(* Logix 5000 project; controller ARS14002_PLC vendor 1 type 14 code 218 rev 30.11; software revision 30.01; part 6 of 13 *)
(* tags used below, declared in another part *)
   ARS_COLLECT : BOOL;
   ARS_COLLECT_AUTO : BOOL;
   ARS_DERIME_AUTO : BOOL;
   AT2_PLANT_ATOMIZING : BOOL;
   AT2_PLANT_BACKFILL : BOOL;
   AT2_PLANT_COLLECT_AUTO : BOOL;
   AT3_PLANT_ATOMIZING : BOOL;
   AT3_PLANT_BACKFILL : BOOL;
   AT3_PLANT_COLLECT_AUTO : BOOL;
   BACKFILL_PAUSE_BLOWBACK_ONS : BOOL;
   BLOWBACK_COMMAND : BOOL;
   BLOWBACK_COUNTER : COUNTER;
   BLOWBACK_PRESS_SPH : REAL;
   BLOWBACK_PRESS_SPL : REAL;
   BLOWBACK_PRESS_UNSAFE : REAL;
   BLOWBACK_REQUEST : BOOL;
   BLOWBACK_REQUEST_OFF_ONS : BOOL;
   BLOWBACK_REQUEST_ONS : BOOL;
   BLOWBACKS_REQUESTED : DINT;
   CALC_NEXT_MONTH_OSR_OB : BOOL;
   COLDBOX_IDLE : BOOL;
   COLDBOX_STANDBY : BOOL;
   Collect_Stop_Dew_Pt : BOOL;
   Collect_Stop_O2 : BOOL;
   FCV_101A : CM_AO_VLV;
   FCV_101B : CM_AO_VLV;
   FCV_101C : CM_AO_VLV;
   FCV_202 : CM_AO_VLV;
   FCV_202_BLOWBACK_POS : REAL;
   FCV_202_OPEN_DLA_PILOT_ADJ : DINT;
   FCV_202_OPEN_DLA_SEC : REAL;
   FCV_202_OPEN_DLA_TMR : TIMER;
   FCV_202_OPEN_INIT : TIMER;
   FCV_202_PVSWITCH : BOOL;   // 0 = PIT-201 1 = PIT-101C
   FCV_202_STARTPOS : REAL;
   FCV_204_ATOMIZE_INIT : TIMER;
   FCV_207_BLOWOFF : BOOL;
   FCV_207_FRONT_END_RESCUE : BOOL;
   FCV_207_FRONT_END_RESCUE_AUTO : BOOL;
   FCV_207_FRONT_END_RESCUE_SP : REAL;
   FCV_207_POSTHEAT_OFF : BOOL;   // Turn off 207 post heat pressurizing
   FCV_207_POSTHEATPRESSURE : REAL;
   FCV_207_POSTHEATPRESSURE_DB : REAL;
   FCV_207_PRESSRELIEF_SPH : REAL;
   FCV_207_PRESSRELIEF_SPL : REAL;
   FCV_207_STATICPOS : REAL;
   FCV_504_LOWPRESS_MAXOPEN : REAL;
   FCV_504_PT_603_LOLOALM : BOOL;
   FCV_504_PT_603_LOWALM : BOOL;
   FCV_504_PT_603_LOWLIM : REAL;
   FCV_504_PT_603_LOWLIM_RESET : REAL;
   FCV_504_SP_Atomize : REAL;
   FCV_504_SP_Atomize_2Tower : REAL;
   FCV_504_SP_Atomize_2Tower_AR : REAL;
   FCV_504_SP_Atomize_2Tower_AR_CALC : REAL;
   FCV_504_SP_Atomize_2Tower_CALC : REAL;
   FCV_504_SP_Atomize_AR : REAL;
   FCV_504_SP_Atomize_AR_CALC : REAL;   // Setpoint with an adjustment for the Pilot Plant
   FCV_504_SP_Atomize_AR_PILOT_ADJ : REAL;   // Adjustment for the atomize setpoint on top of what it would be for normal furnaces
   FCV_504_SP_Atomize_CALC : REAL;
   FCV_504_SP_Atomize_FRONT_END : REAL;
   FCV_504_SP_Atomize_PILOT_ADJ : REAL;
   FCV_504_SP_Idle : REAL;
   FCV_504_SP_Idle_AR : REAL;
   FCV_504_SP_Idle_AR_STORAGE : REAL;
   FCV_504_SP_Idle_STORAGE : REAL;
   FCV_504_SP_Standby : REAL;
   FCV_504_SP_Standby_AR : REAL;
   FCV_504_STARTPOS : REAL;
   FCV_603_Atomize_Start_CV : REAL;
   FCV_603_BUMP_TMR : TIMER;
   FCV_603_SP_Atomize : REAL;
   FCV_603_SP_Idle : REAL;
   FCV_603_SP_Standby : REAL;
   MODE_ATOMIZE : BOOL;
   MODE_IDLE : BOOL;
   MODE_STANDBY_IDLE : BOOL;
   MODE_STANDBY_PUMPUP : BOOL;
   PDT_603 : CM_AI_SCL_ALT;
   PDT_701 : CM_AI_SCL_ALT;
   PIDE_202 : PID_ENHANCED;
   PIDE_204 : PID_ENHANCED;
   PIDE_207 : PID_ENHANCED;
   PIDE_504 : PID_ENHANCED;
   PIDE_504_FRONT_END_CONTROL : BOOL;
   PIDE_504_FRONT_END_CONTROL_REQUEST : BOOL;
   PIDE_504_MODE : BOOL;   // 0 = Argon (PT-601) 1 = N2 (PT-603)
   PIDE_603 : PID_ENHANCED;
   PIDE_603_CVLimit_TON : TIMER;
   PIDE_603_CVLimitLOW_TON : TIMER;
   PIDE_605 : PID_ENHANCED;
   Pilot_Atomizing_Valve_Close_TON : TIMER;
   Pilot_Atomizing_Valve_Open_TON : TIMER;
   Pilot_Inlet_Valve_Open_TON : TIMER;
   PILOT_PLANT_ATOMIZING : BOOL;
   PILOT_PLANT_BACKFILL : BOOL;
   PILOT_PLANT_COLLECT_AUTO : BOOL;
   PT_1002 : CM_AI_SCL;
   PT_101C : CM_AI_SCL;
   PT_201 : CM_AI_SCL;
   PT_222 : CM_AI_SCL;
   PT_601 : CM_AI_SCL;
   PT_601_FCV_202_SP : REAL;
   PT_601_LR : CM_AI_SCL;
   PT_603 : CM_AI_SCL;
   Pull_Hold : BOOL;
   PWHMI_Post_Atomize_TMR : TIMER;
   SV_202F : CM_DO_GENERIC;
   SV_205 : CM_DO_GENERIC;
   SV_205_FIXED : BOOL;
   SV_205_Pressure_SPH : REAL;
   SV_205_Pressure_SPH_TEST : REAL;
   SV_205_Pressure_SPL : REAL;
   SV_205_Pressure_SPL_TEST : REAL;
   SV_207F : CM_DO_GENERIC;
   SV_221X : CM_DO_GENERIC;
   SV_221X_ONS : BOOL;
   SV_504F : CM_DO_GENERIC;
   SV_505X : CM_DO_GENERIC;
   SV_603F : CM_DO_GENERIC;
   SV_605F : CM_DO_GENERIC;
   TE_501 : CM_AI_SCL;
   TE_501_MIN_SV_202 : REAL;
   TE_902 : CM_AI_SCL;
   TimeStamp : DINT[7];
   TK_220_FILLS_MONTH : COUNTER;
   TK_220_Pressure_SPH : INT;
   TK_220_Pressure_SPL : INT;
   TK_700_Full : BOOL;
   TK_700_FULL_DLA_TMR : TIMER;
   TK_700_Full_SPH : REAL;
   TK_700_Full_SPL : REAL;
   TK_700_Low : BOOL;
   TK_700_LOW_DLA_TMR : TIMER;
   TK_700_Low_SPH : REAL;
   TK_700_Low_SPL : REAL;
   TK_700_NOT_FULL_DLA_TMR : TIMER;
   TK_700_OVERFULL_DLA_TMR : TIMER;
   XV_505_PT_603_SPH_VENT : REAL;
   XV_505_PT_603_SPL_VENT : REAL;
(* MainProgram, continued *)

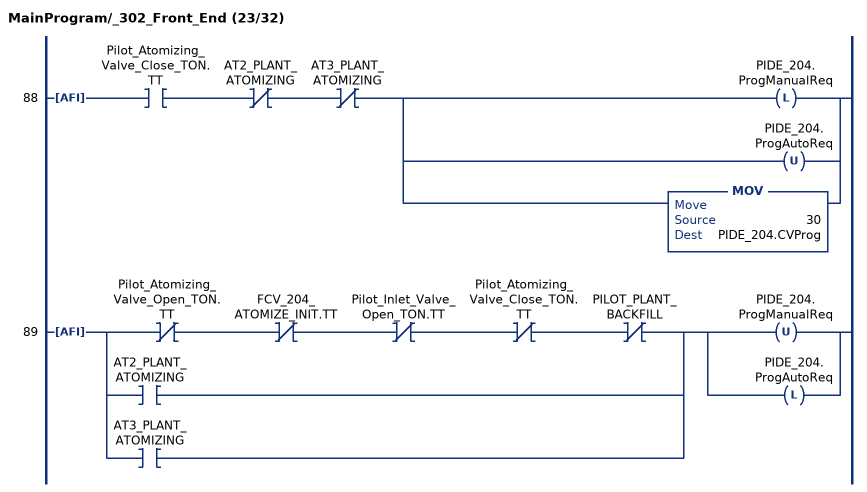
   [picture p107: MainProgram/_302_Front_End rungs 88-89]
   88: AFI()XIC(Pilot_Atomizing_Valve_Close_TON.TT)XIO(AT2_PLANT_ATOMIZING)XIO(AT3_PLANT_ATOMIZING)[OTL(PIDE_204.ProgManualReq) ,OTU(PIDE_204.ProgAutoReq) ,MOV(30,PIDE_204.CVProg) ];
   89: AFI()[XIO(Pilot_Atomizing_Valve_Open_TON.TT) XIO(FCV_204_ATOMIZE_INIT.TT) XIO(Pilot_Inlet_Valve_Open_TON.TT) XIO(Pilot_Atomizing_Valve_Close_TON.TT) XIO(PILOT_PLANT_BACKFILL) ,XIC(AT2_PLANT_ATOMIZING) ,XIC(AT3_PLANT_ATOMIZING) ][OTU(PIDE_204.ProgManualReq) ,OTL(PIDE_204.ProgAutoReq) ];
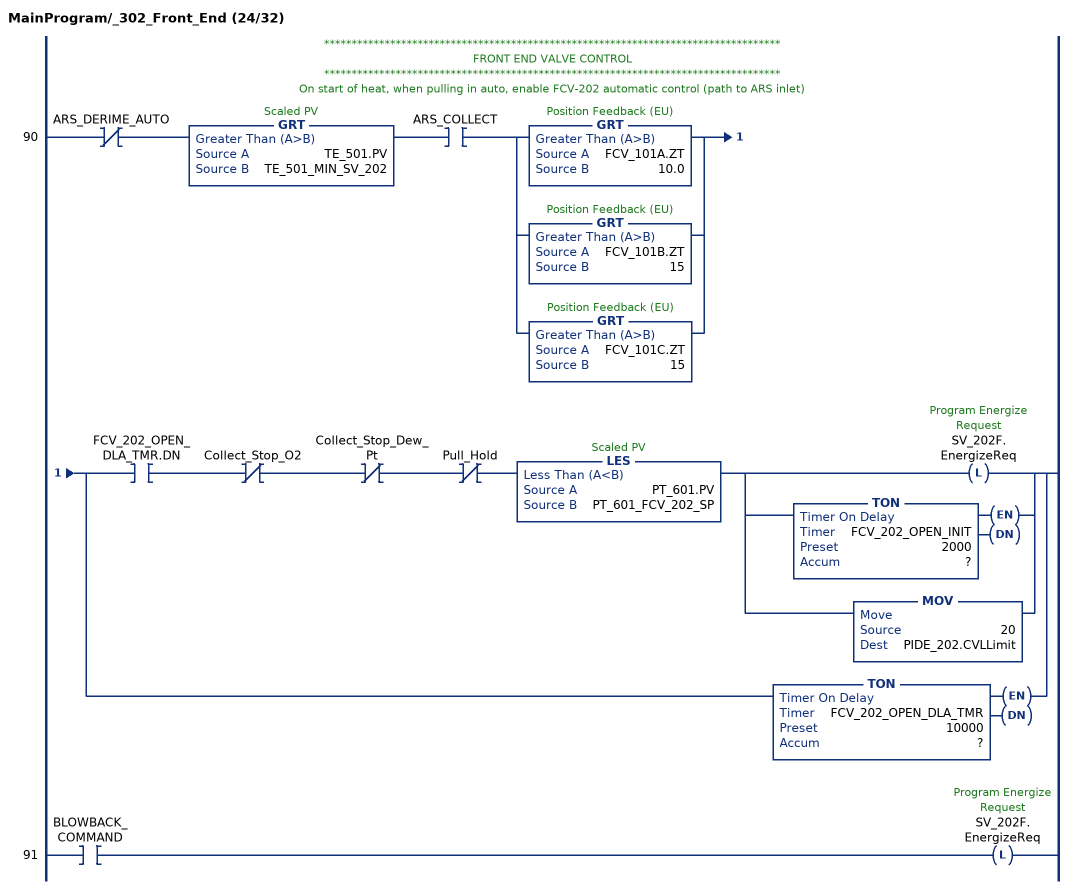
   // ***********************************************************************************
   // FRONT END VALVE CONTROL
   // ***********************************************************************************
   // On start of heat, when pulling in auto, enable FCV-202 automatic control (path to ARS inlet)
   90: XIO(ARS_DERIME_AUTO)GRT(TE_501.PV,TE_501_MIN_SV_202)XIC(ARS_COLLECT)[GRT(FCV_101A.ZT,10.0) ,GRT(FCV_101B.ZT,15) ,GRT(FCV_101C.ZT,15) ][XIC(FCV_202_OPEN_DLA_TMR.DN) XIO(Collect_Stop_O2) XIO(Collect_Stop_Dew_Pt) XIO(Pull_Hold) LES(PT_601.PV,PT_601_FCV_202_SP) [OTL(SV_202F.EnergizeReq) ,TON(FCV_202_OPEN_INIT,?,?) ,MOV(20,PIDE_202.CVLLimit) ] ,TON(FCV_202_OPEN_DLA_TMR,?,?) ];
   91: XIC(BLOWBACK_COMMAND)OTL(SV_202F.EnergizeReq);
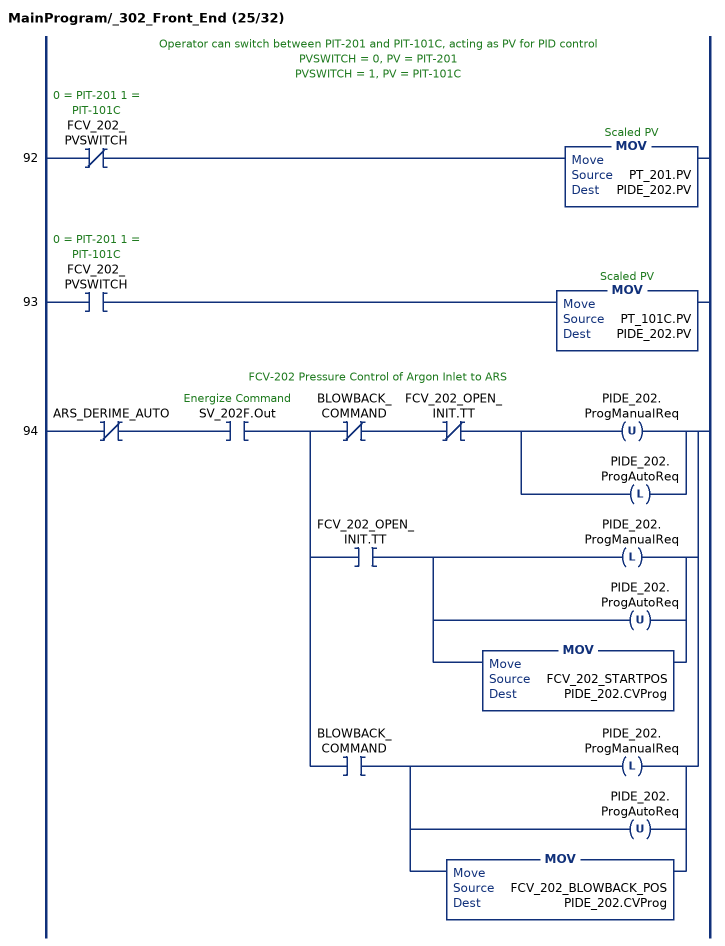
   // Operator can switch between PIT-201 and PIT-101C, acting as PV for PID control
   // PVSWITCH = 0, PV = PIT-201
   // PVSWITCH = 1, PV = PIT-101C
   92: XIO(FCV_202_PVSWITCH)MOV(PT_201.PV,PIDE_202.PV);
   93: XIC(FCV_202_PVSWITCH)MOV(PT_101C.PV,PIDE_202.PV);
   // FCV-202 Pressure Control of Argon Inlet to ARS
   94: XIO(ARS_DERIME_AUTO)XIC(SV_202F.Out)[XIO(BLOWBACK_COMMAND) XIO(FCV_202_OPEN_INIT.TT) [OTU(PIDE_202.ProgManualReq) ,OTL(PIDE_202.ProgAutoReq) ] ,XIC(FCV_202_OPEN_INIT.TT) [OTL(PIDE_202.ProgManualReq) ,OTU(PIDE_202.ProgAutoReq) ,MOV(FCV_202_STARTPOS,PIDE_202.CVProg) ] ,XIC(BLOWBACK_COMMAND) [OTL(PIDE_202.ProgManualReq) ,OTU(PIDE_202.ProgAutoReq) ,MOV(FCV_202_BLOWBACK_POS,PIDE_202.CVProg) ] ];
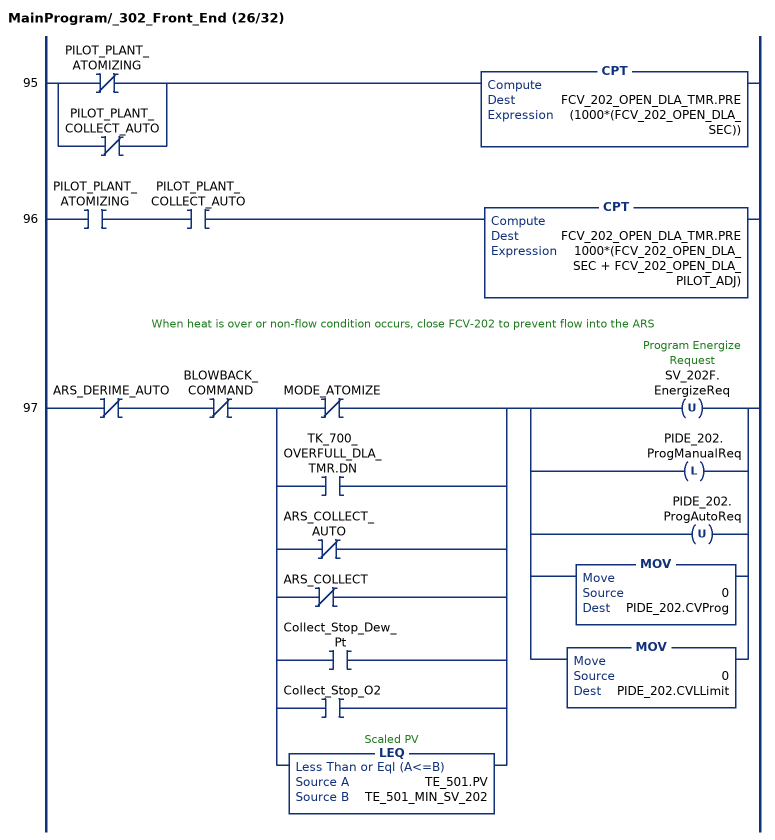
   95: [XIO(PILOT_PLANT_ATOMIZING) ,XIO(PILOT_PLANT_COLLECT_AUTO) ]CPT(FCV_202_OPEN_DLA_TMR.PRE,(1000*(FCV_202_OPEN_DLA_SEC)));
   96: XIC(PILOT_PLANT_ATOMIZING)XIC(PILOT_PLANT_COLLECT_AUTO)CPT(FCV_202_OPEN_DLA_TMR.PRE,1000*(FCV_202_OPEN_DLA_SEC + FCV_202_OPEN_DLA_PILOT_ADJ));
   // When heat is over or non-flow condition occurs, close FCV-202 to prevent flow into the ARS
   97: XIO(ARS_DERIME_AUTO)XIO(BLOWBACK_COMMAND)[XIO(MODE_ATOMIZE) ,XIC(TK_700_OVERFULL_DLA_TMR.DN) ,XIO(ARS_COLLECT_AUTO) ,XIO(ARS_COLLECT) ,XIC(Collect_Stop_Dew_Pt) ,XIC(Collect_Stop_O2) ,LEQ(TE_501.PV,TE_501_MIN_SV_202) ][OTU(SV_202F.EnergizeReq) ,OTL(PIDE_202.ProgManualReq) ,OTU(PIDE_202.ProgAutoReq) ,MOV(0,PIDE_202.CVProg) ,MOV(0,PIDE_202.CVLLimit) ];
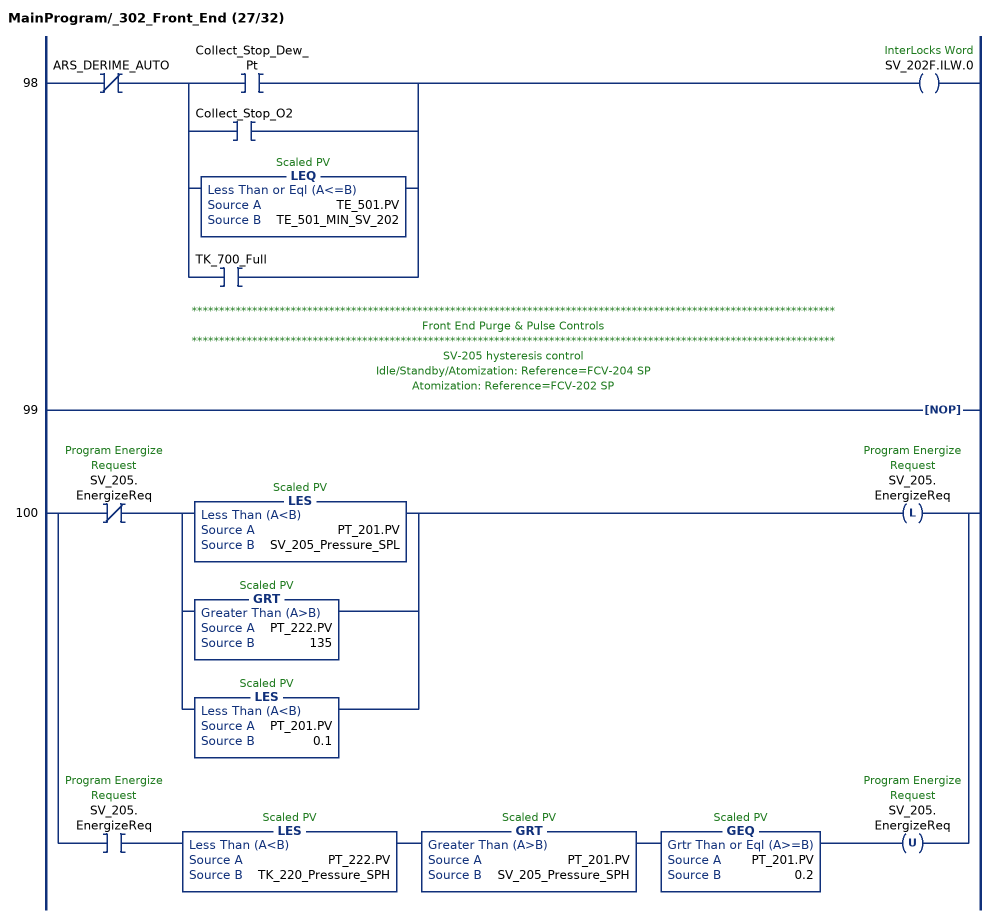
   98: XIO(ARS_DERIME_AUTO)[XIC(Collect_Stop_Dew_Pt) ,XIC(Collect_Stop_O2) ,LEQ(TE_501.PV,TE_501_MIN_SV_202) ,XIC(TK_700_Full) ]OTE(SV_202F.ILW.0);
   // *********************************************************************************************************************
   // Front End Purge & Pulse Controls
   // *********************************************************************************************************************
   // SV-205 hysteresis control
   // Idle/Standby/Atomization: Reference=FCV-204 SP
   // Atomization: Reference=FCV-202 SP
   99: NOP();
   100: [XIO(SV_205.EnergizeReq) [LES(PT_201.PV,SV_205_Pressure_SPL) ,GRT(PT_222.PV,135) ,LES(PT_201.PV,0.1) ] OTL(SV_205.EnergizeReq) ,XIC(SV_205.EnergizeReq) LES(PT_222.PV,TK_220_Pressure_SPH) GRT(PT_201.PV,SV_205_Pressure_SPH) GEQ(PT_201.PV,0.2) OTU(SV_205.EnergizeReq) ];
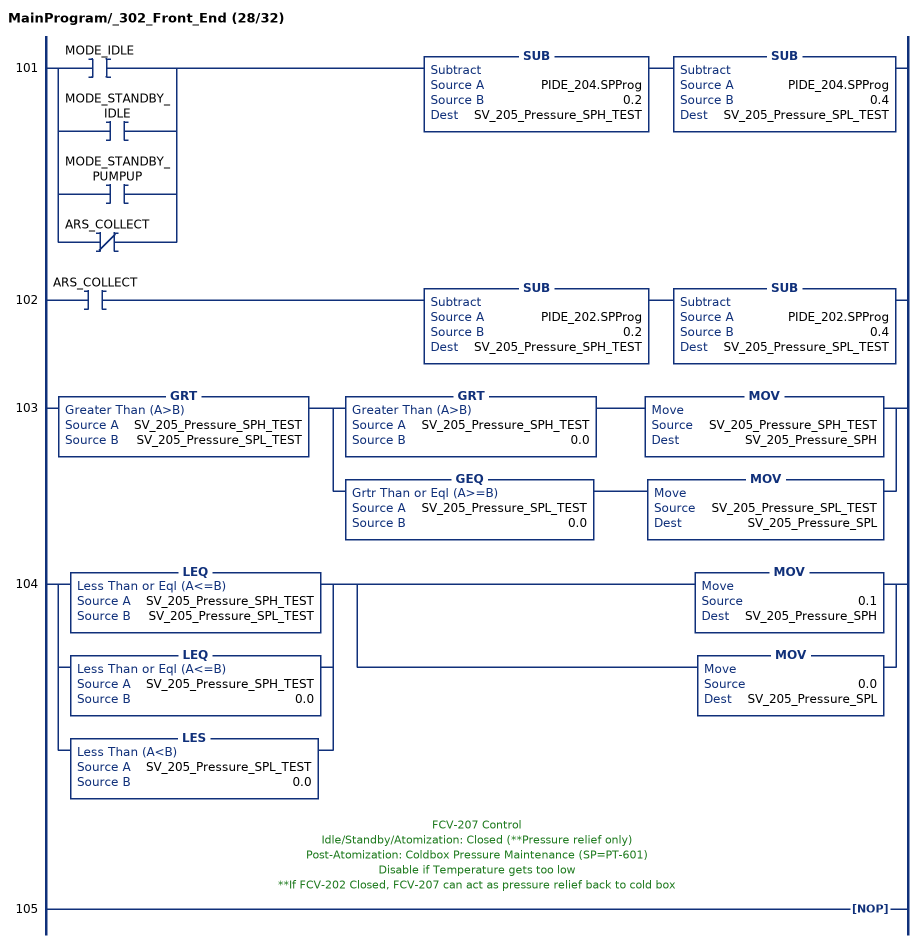
   101: [XIC(MODE_IDLE) ,XIC(MODE_STANDBY_IDLE) ,XIC(MODE_STANDBY_PUMPUP) ,XIO(ARS_COLLECT) ]SUB(PIDE_204.SPProg,0.2,SV_205_Pressure_SPH_TEST)SUB(PIDE_204.SPProg,0.4,SV_205_Pressure_SPL_TEST);
   102: XIC(ARS_COLLECT)SUB(PIDE_202.SPProg,0.2,SV_205_Pressure_SPH_TEST)SUB(PIDE_202.SPProg,0.4,SV_205_Pressure_SPL_TEST);
   103: GRT(SV_205_Pressure_SPH_TEST,SV_205_Pressure_SPL_TEST)[GRT(SV_205_Pressure_SPH_TEST,0.0) MOV(SV_205_Pressure_SPH_TEST,SV_205_Pressure_SPH) ,GEQ(SV_205_Pressure_SPL_TEST,0.0) MOV(SV_205_Pressure_SPL_TEST,SV_205_Pressure_SPL) ];
   104: [LEQ(SV_205_Pressure_SPH_TEST,SV_205_Pressure_SPL_TEST) ,LEQ(SV_205_Pressure_SPH_TEST,0.0) ,LES(SV_205_Pressure_SPL_TEST,0.0) ][MOV(0.1,SV_205_Pressure_SPH) ,MOV(0.0,SV_205_Pressure_SPL) ];
   // FCV-207 Control
   // Idle/Standby/Atomization: Closed (**Pressure relief only)
   // Post-Atomization: Coldbox Pressure Maintenance (SP=PT-601)
   // Disable if Temperature gets too low
   // **If FCV-202 Closed, FCV-207 can act as pressure relief back to cold box
   105: NOP();
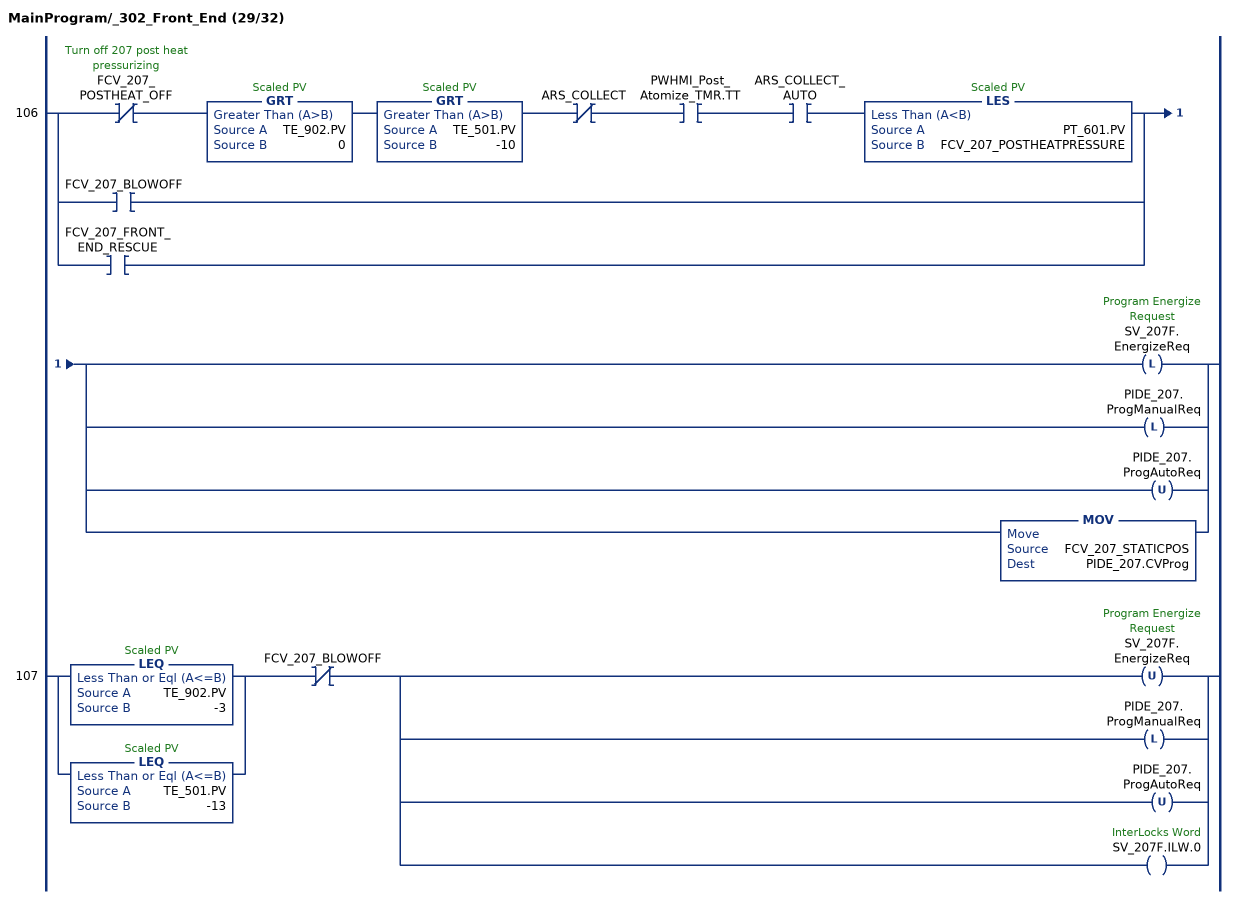
   106: [XIO(FCV_207_POSTHEAT_OFF) GRT(TE_902.PV,0) GRT(TE_501.PV,-10) XIO(ARS_COLLECT) XIC(PWHMI_Post_Atomize_TMR.TT) XIC(ARS_COLLECT_AUTO) LES(PT_601.PV,FCV_207_POSTHEATPRESSURE) ,XIC(FCV_207_BLOWOFF) ,XIC(FCV_207_FRONT_END_RESCUE) ][OTL(SV_207F.EnergizeReq) ,OTL(PIDE_207.ProgManualReq) ,OTU(PIDE_207.ProgAutoReq) ,MOV(FCV_207_STATICPOS,PIDE_207.CVProg) ];
   107: [LEQ(TE_902.PV,-3) ,LEQ(TE_501.PV,-13) ]XIO(FCV_207_BLOWOFF)[OTU(SV_207F.EnergizeReq) ,OTL(PIDE_207.ProgManualReq) ,OTU(PIDE_207.ProgAutoReq) ,OTE(SV_207F.ILW.0) ];
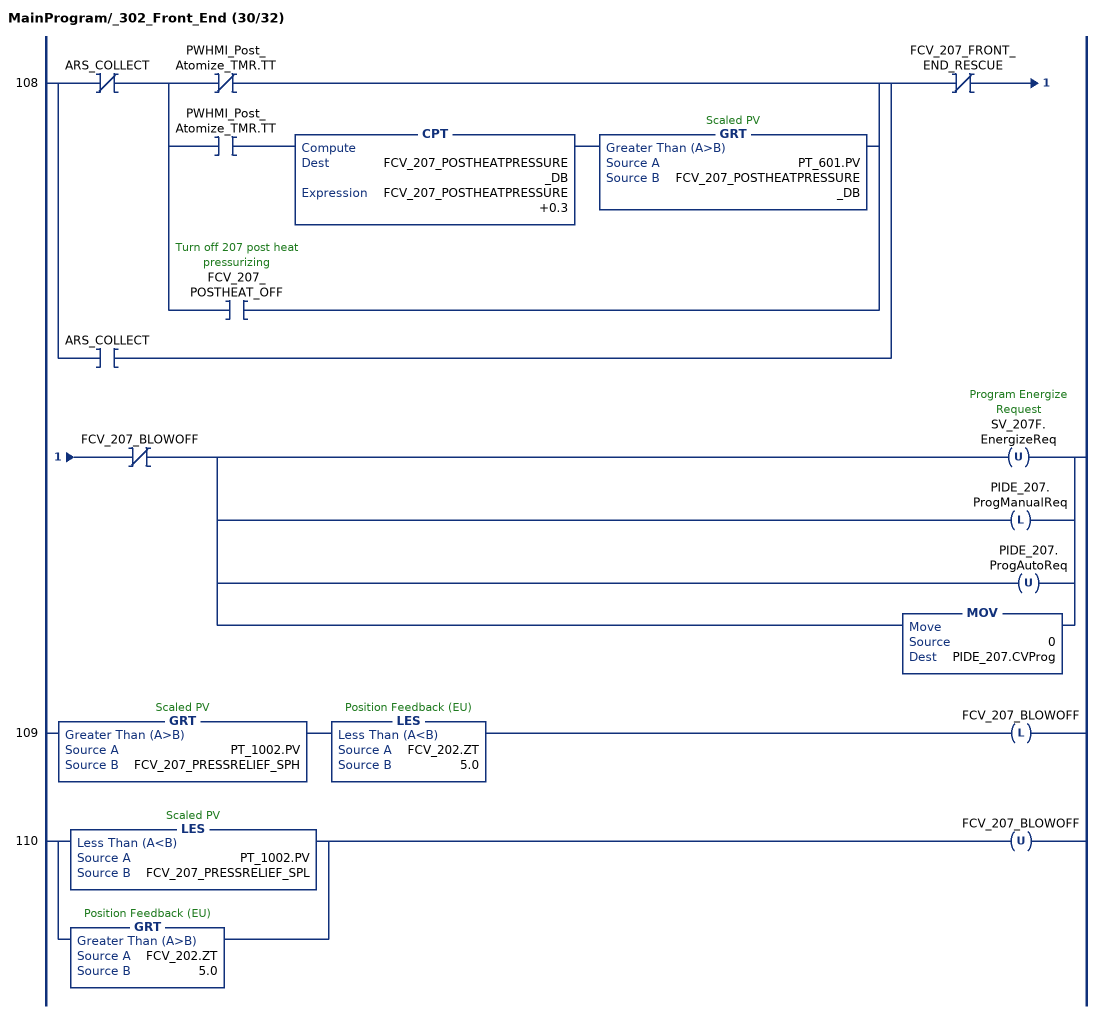
   108: [XIO(ARS_COLLECT) [XIO(PWHMI_Post_Atomize_TMR.TT) ,XIC(PWHMI_Post_Atomize_TMR.TT) CPT(FCV_207_POSTHEATPRESSURE_DB,FCV_207_POSTHEATPRESSURE+0.3) GRT(PT_601.PV,FCV_207_POSTHEATPRESSURE_DB) ,XIC(FCV_207_POSTHEAT_OFF) ] ,XIC(ARS_COLLECT) ]XIO(FCV_207_FRONT_END_RESCUE)XIO(FCV_207_BLOWOFF)[OTU(SV_207F.EnergizeReq) ,OTL(PIDE_207.ProgManualReq) ,OTU(PIDE_207.ProgAutoReq) ,MOV(0,PIDE_207.CVProg) ];
   109: GRT(PT_1002.PV,FCV_207_PRESSRELIEF_SPH)LES(FCV_202.ZT,5.0)OTL(FCV_207_BLOWOFF);
   110: [LES(PT_1002.PV,FCV_207_PRESSRELIEF_SPL) ,GRT(FCV_202.ZT,5.0) ]OTU(FCV_207_BLOWOFF);
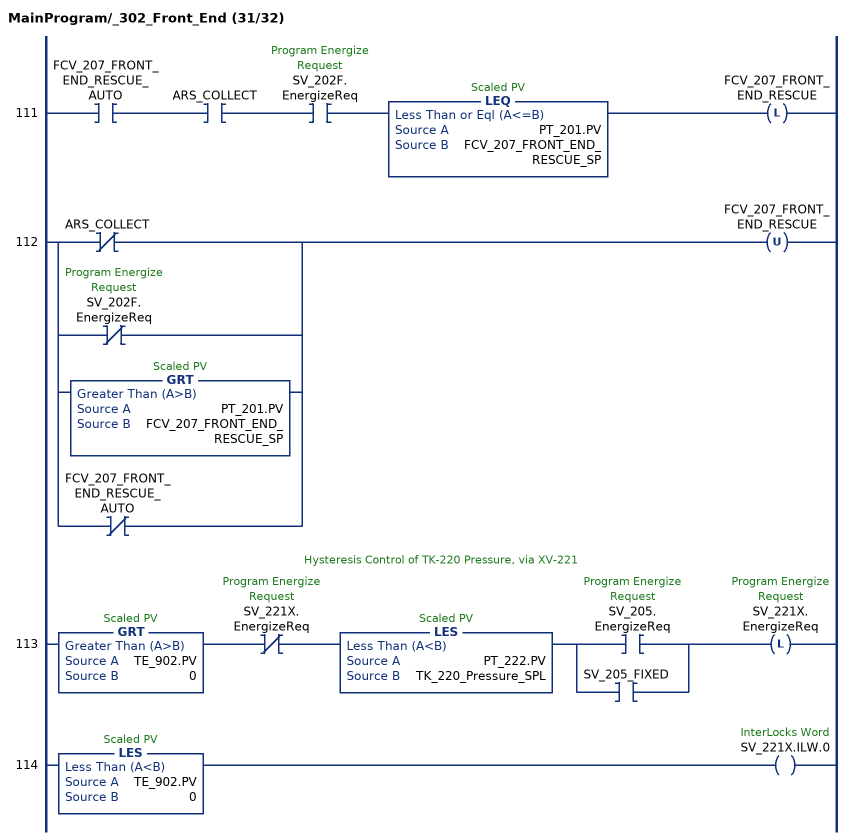
   111: XIC(FCV_207_FRONT_END_RESCUE_AUTO)XIC(ARS_COLLECT)XIC(SV_202F.EnergizeReq)LEQ(PT_201.PV,FCV_207_FRONT_END_RESCUE_SP)OTL(FCV_207_FRONT_END_RESCUE);
   112: [XIO(ARS_COLLECT) ,XIO(SV_202F.EnergizeReq) ,GRT(PT_201.PV,FCV_207_FRONT_END_RESCUE_SP) ,XIO(FCV_207_FRONT_END_RESCUE_AUTO) ]OTU(FCV_207_FRONT_END_RESCUE);
   // Hysteresis Control of TK-220 Pressure, via XV-221
   113: GRT(TE_902.PV,0)XIO(SV_221X.EnergizeReq)LES(PT_222.PV,TK_220_Pressure_SPL)[XIC(SV_205.EnergizeReq) ,XIC(SV_205_FIXED) ]OTL(SV_221X.EnergizeReq);
   114: LES(TE_902.PV,0)OTE(SV_221X.ILW.0);
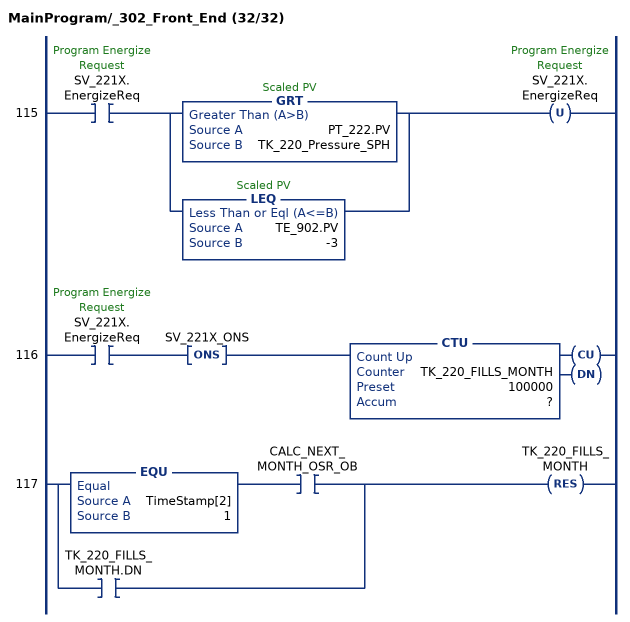
   115: XIC(SV_221X.EnergizeReq)[GRT(PT_222.PV,TK_220_Pressure_SPH) ,LEQ(TE_902.PV,-3) ]OTU(SV_221X.EnergizeReq);
   116: XIC(SV_221X.EnergizeReq)ONS(SV_221X_ONS)CTU(TK_220_FILLS_MONTH,?,?);
   117: [EQU(TimeStamp[2],1) XIC(CALC_NEXT_MONTH_OSR_OB) ,XIC(TK_220_FILLS_MONTH.DN) ]RES(TK_220_FILLS_MONTH);
END_ROUTINE

ROUTINE _303_Cold_Box   (* ladder *)
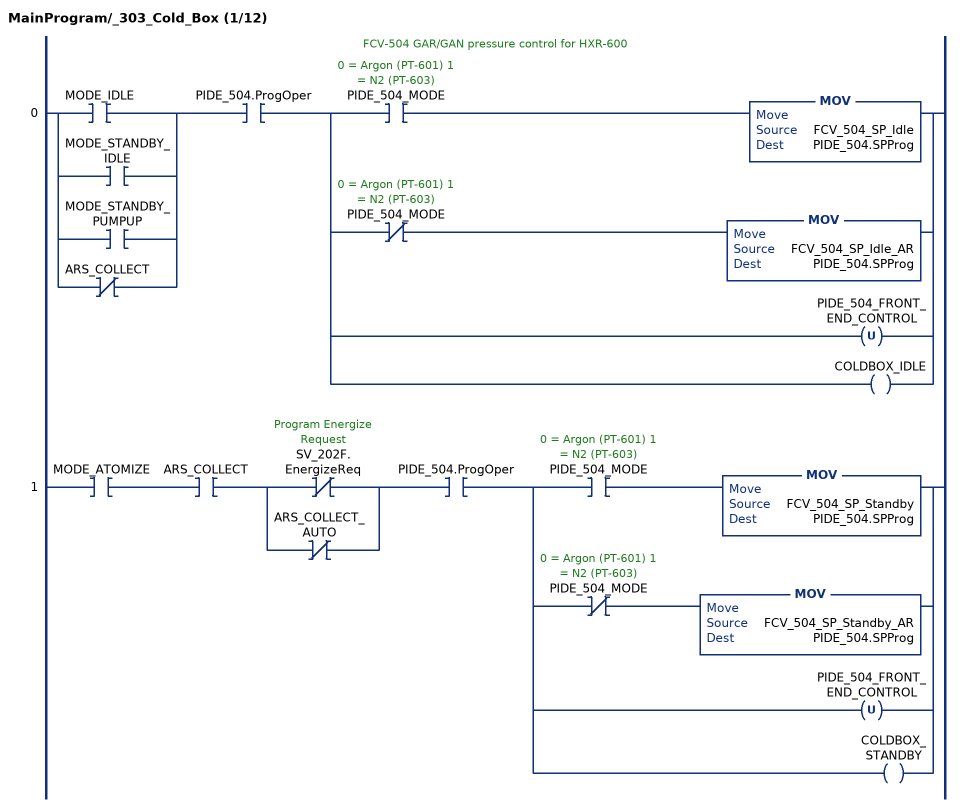
   // FCV-504 GAR/GAN pressure control for HXR-600
   0: [XIC(MODE_IDLE) ,XIC(MODE_STANDBY_IDLE) ,XIC(MODE_STANDBY_PUMPUP) ,XIO(ARS_COLLECT) ]XIC(PIDE_504.ProgOper)[XIC(PIDE_504_MODE) MOV(FCV_504_SP_Idle,PIDE_504.SPProg) ,XIO(PIDE_504_MODE) MOV(FCV_504_SP_Idle_AR,PIDE_504.SPProg) ,OTU(PIDE_504_FRONT_END_CONTROL) ,OTE(COLDBOX_IDLE) ];
   1: XIC(MODE_ATOMIZE)XIC(ARS_COLLECT)[XIO(SV_202F.EnergizeReq) ,XIO(ARS_COLLECT_AUTO) ]XIC(PIDE_504.ProgOper)[XIC(PIDE_504_MODE) MOV(FCV_504_SP_Standby,PIDE_504.SPProg) ,XIO(PIDE_504_MODE) MOV(FCV_504_SP_Standby_AR,PIDE_504.SPProg) ,OTU(PIDE_504_FRONT_END_CONTROL) ,OTE(COLDBOX_STANDBY) ];
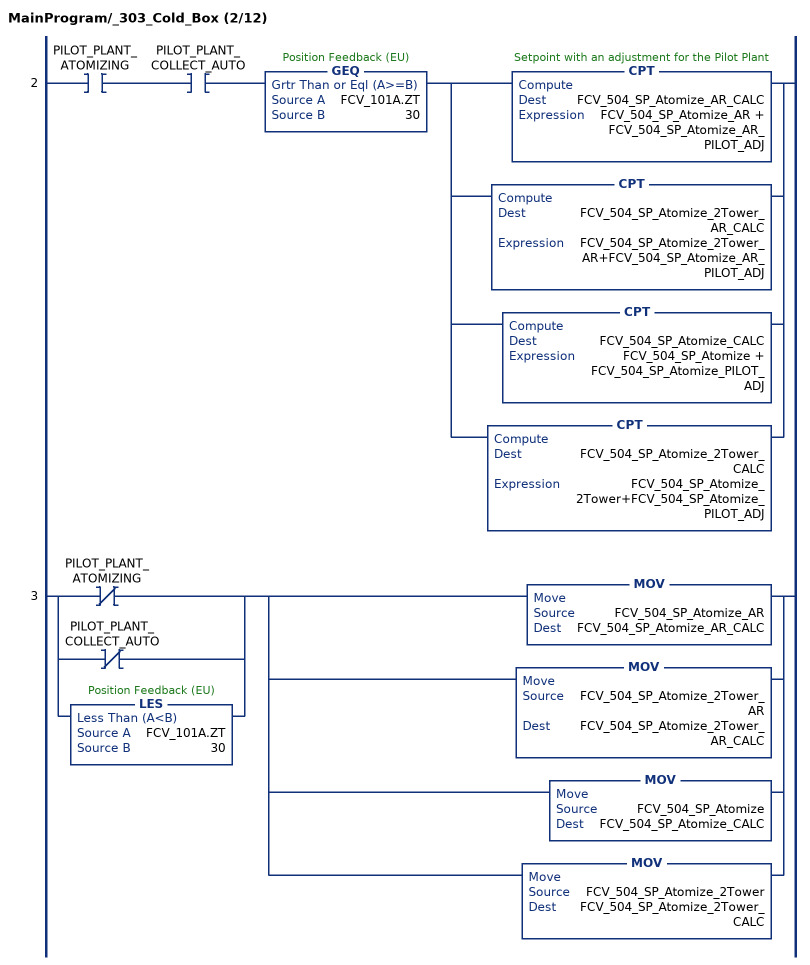
   2: XIC(PILOT_PLANT_ATOMIZING)XIC(PILOT_PLANT_COLLECT_AUTO)GEQ(FCV_101A.ZT,30)[CPT(FCV_504_SP_Atomize_AR_CALC,FCV_504_SP_Atomize_AR + FCV_504_SP_Atomize_AR_PILOT_ADJ) ,CPT(FCV_504_SP_Atomize_2Tower_AR_CALC,FCV_504_SP_Atomize_2Tower_AR+FCV_504_SP_Atomize_AR_PILOT_ADJ) ,CPT(FCV_504_SP_Atomize_CALC,FCV_504_SP_Atomize + FCV_504_SP_Atomize_PILOT_ADJ) ,CPT(FCV_504_SP_Atomize_2Tower_CALC,FCV_504_SP_Atomize_2Tower+FCV_504_SP_Atomize_PILOT_ADJ) ];
   3: [XIO(PILOT_PLANT_ATOMIZING) ,XIO(PILOT_PLANT_COLLECT_AUTO) ,LES(FCV_101A.ZT,30) ][MOV(FCV_504_SP_Atomize_AR,FCV_504_SP_Atomize_AR_CALC) ,MOV(FCV_504_SP_Atomize_2Tower_AR,FCV_504_SP_Atomize_2Tower_AR_CALC) ,MOV(FCV_504_SP_Atomize,FCV_504_SP_Atomize_CALC) ,MOV(FCV_504_SP_Atomize_2Tower,FCV_504_SP_Atomize_2Tower_CALC) ];
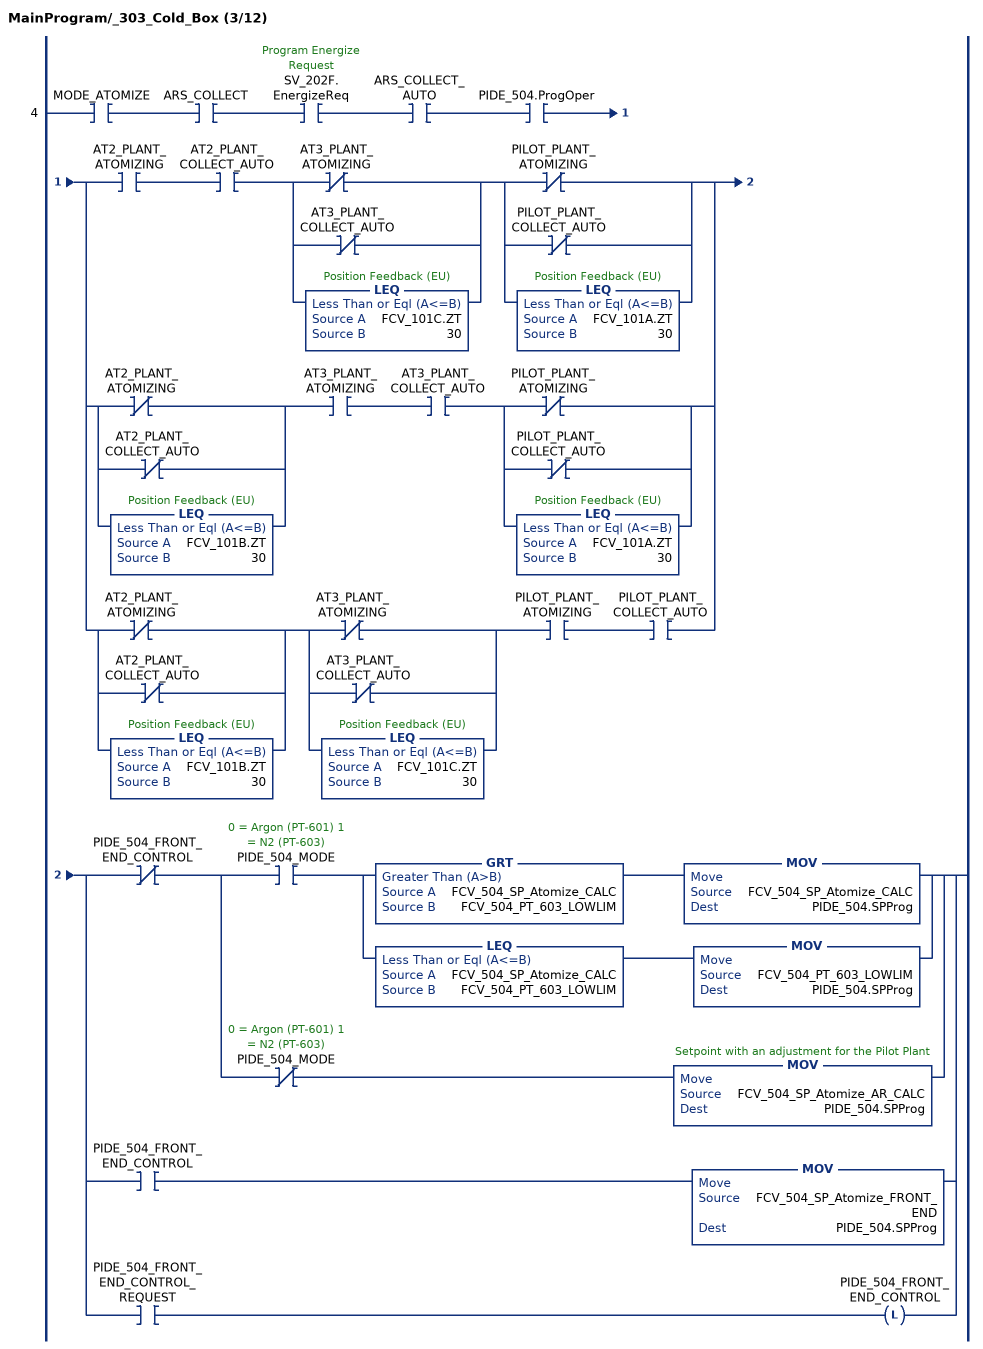
   4: XIC(MODE_ATOMIZE)XIC(ARS_COLLECT)XIC(SV_202F.EnergizeReq)XIC(ARS_COLLECT_AUTO)XIC(PIDE_504.ProgOper)[XIC(AT2_PLANT_ATOMIZING) XIC(AT2_PLANT_COLLECT_AUTO) [XIO(AT3_PLANT_ATOMIZING) ,XIO(AT3_PLANT_COLLECT_AUTO) ,LEQ(FCV_101C.ZT,30) ] [XIO(PILOT_PLANT_ATOMIZING) ,XIO(PILOT_PLANT_COLLECT_AUTO) ,LEQ(FCV_101A.ZT,30) ] ,[XIO(AT2_PLANT_ATOMIZING) ,XIO(AT2_PLANT_COLLECT_AUTO) ,LEQ(FCV_101B.ZT,30) ] XIC(AT3_PLANT_ATOMIZING) XIC(AT3_PLANT_COLLECT_AUTO) [XIO(PILOT_PLANT_ATOMIZING) ,XIO(PILOT_PLANT_COLLECT_AUTO) ,LEQ(FCV_101A.ZT,30) ] ,[XIO(AT2_PLANT_ATOMIZING) ,XIO(AT2_PLANT_COLLECT_AUTO) ,LEQ(FCV_101B.ZT,30) ] [XIO(AT3_PLANT_ATOMIZING) ,XIO(AT3_PLANT_COLLECT_AUTO) ,LEQ(FCV_101C.ZT,30) ] XIC(PILOT_PLANT_ATOMIZING) XIC(PILOT_PLANT_COLLECT_AUTO) ][XIO(PIDE_504_FRONT_END_CONTROL) [XIC(PIDE_504_MODE) [GRT(FCV_504_SP_Atomize_CALC,FCV_504_PT_603_LOWLIM) MOV(FCV_504_SP_Atomize_CALC,PIDE_504.SPProg) ,LEQ(FCV_504_SP_Atomize_CALC,FCV_504_PT_603_LOWLIM) MOV(FCV_504_PT_603_LOWLIM,PIDE_504.SPProg) ] ,XIO(PIDE_504_MODE) MOV(FCV_504_SP_Atomize_AR_CALC,PIDE_504.SPProg) ] ,XIC(PIDE_504_FRONT_END_CONTROL) MOV(FCV_504_SP_Atomize_FRONT_END,PIDE_504.SPProg) ,XIC(PIDE_504_FRONT_END_CONTROL_REQUEST) OTL(PIDE_504_FRONT_END_CONTROL) ];
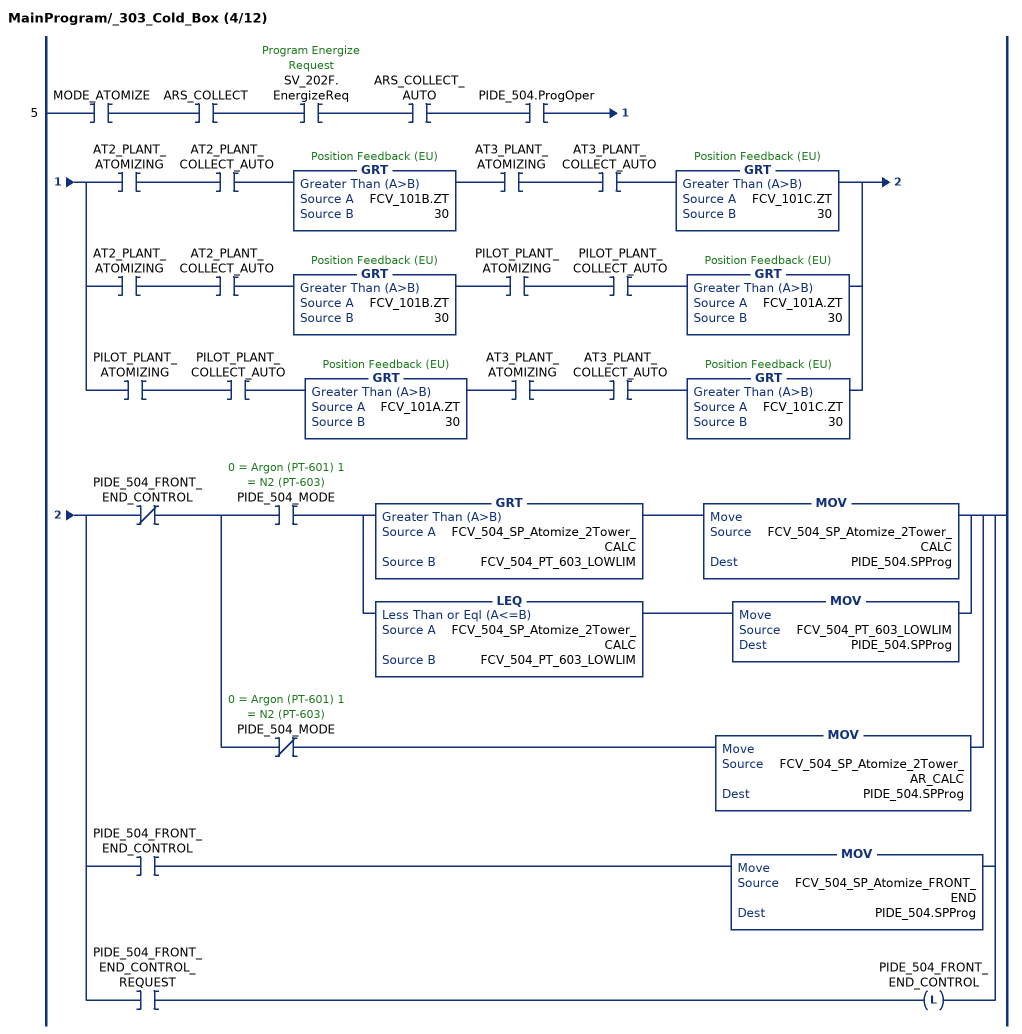
   5: XIC(MODE_ATOMIZE)XIC(ARS_COLLECT)XIC(SV_202F.EnergizeReq)XIC(ARS_COLLECT_AUTO)XIC(PIDE_504.ProgOper)[XIC(AT2_PLANT_ATOMIZING) XIC(AT2_PLANT_COLLECT_AUTO) GRT(FCV_101B.ZT,30) XIC(AT3_PLANT_ATOMIZING) XIC(AT3_PLANT_COLLECT_AUTO) GRT(FCV_101C.ZT,30) ,XIC(AT2_PLANT_ATOMIZING) XIC(AT2_PLANT_COLLECT_AUTO) GRT(FCV_101B.ZT,30) XIC(PILOT_PLANT_ATOMIZING) XIC(PILOT_PLANT_COLLECT_AUTO) GRT(FCV_101A.ZT,30) ,XIC(PILOT_PLANT_ATOMIZING) XIC(PILOT_PLANT_COLLECT_AUTO) GRT(FCV_101A.ZT,30) XIC(AT3_PLANT_ATOMIZING) XIC(AT3_PLANT_COLLECT_AUTO) GRT(FCV_101C.ZT,30) ][XIO(PIDE_504_FRONT_END_CONTROL) [XIC(PIDE_504_MODE) [GRT(FCV_504_SP_Atomize_2Tower_CALC,FCV_504_PT_603_LOWLIM) MOV(FCV_504_SP_Atomize_2Tower_CALC,PIDE_504.SPProg) ,LEQ(FCV_504_SP_Atomize_2Tower_CALC,FCV_504_PT_603_LOWLIM) MOV(FCV_504_PT_603_LOWLIM,PIDE_504.SPProg) ] ,XIO(PIDE_504_MODE) MOV(FCV_504_SP_Atomize_2Tower_AR_CALC,PIDE_504.SPProg) ] ,XIC(PIDE_504_FRONT_END_CONTROL) MOV(FCV_504_SP_Atomize_FRONT_END,PIDE_504.SPProg) ,XIC(PIDE_504_FRONT_END_CONTROL_REQUEST) OTL(PIDE_504_FRONT_END_CONTROL) ];
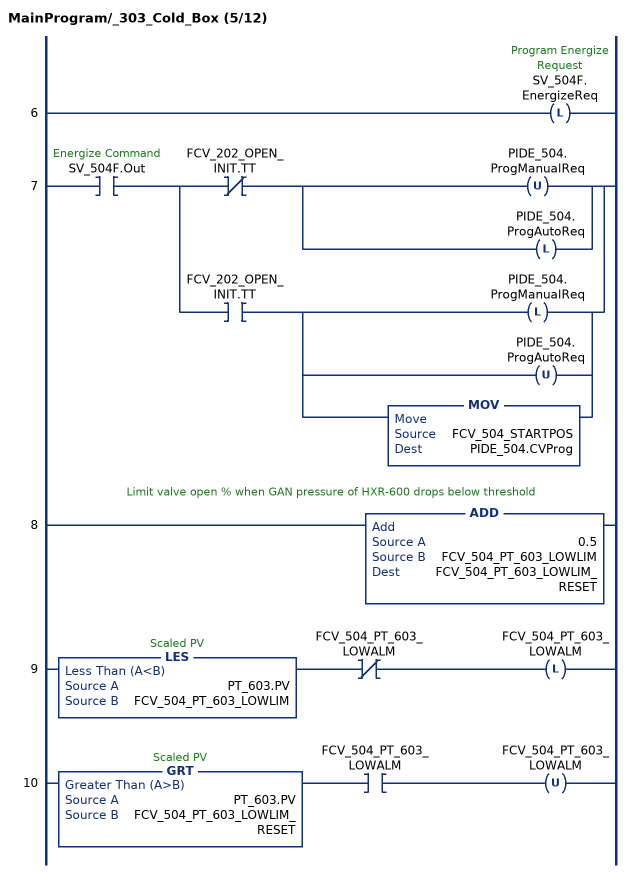
   6: OTL(SV_504F.EnergizeReq);
   7: XIC(SV_504F.Out)[XIO(FCV_202_OPEN_INIT.TT) [OTU(PIDE_504.ProgManualReq) ,OTL(PIDE_504.ProgAutoReq) ] ,XIC(FCV_202_OPEN_INIT.TT) [OTL(PIDE_504.ProgManualReq) ,OTU(PIDE_504.ProgAutoReq) ,MOV(FCV_504_STARTPOS,PIDE_504.CVProg) ] ];
   // Limit valve open % when GAN pressure of HXR-600 drops below threshold
   8: ADD(0.5,FCV_504_PT_603_LOWLIM,FCV_504_PT_603_LOWLIM_RESET);
   9: LES(PT_603.PV,FCV_504_PT_603_LOWLIM)XIO(FCV_504_PT_603_LOWALM)OTL(FCV_504_PT_603_LOWALM);
   10: GRT(PT_603.PV,FCV_504_PT_603_LOWLIM_RESET)XIC(FCV_504_PT_603_LOWALM)OTU(FCV_504_PT_603_LOWALM);
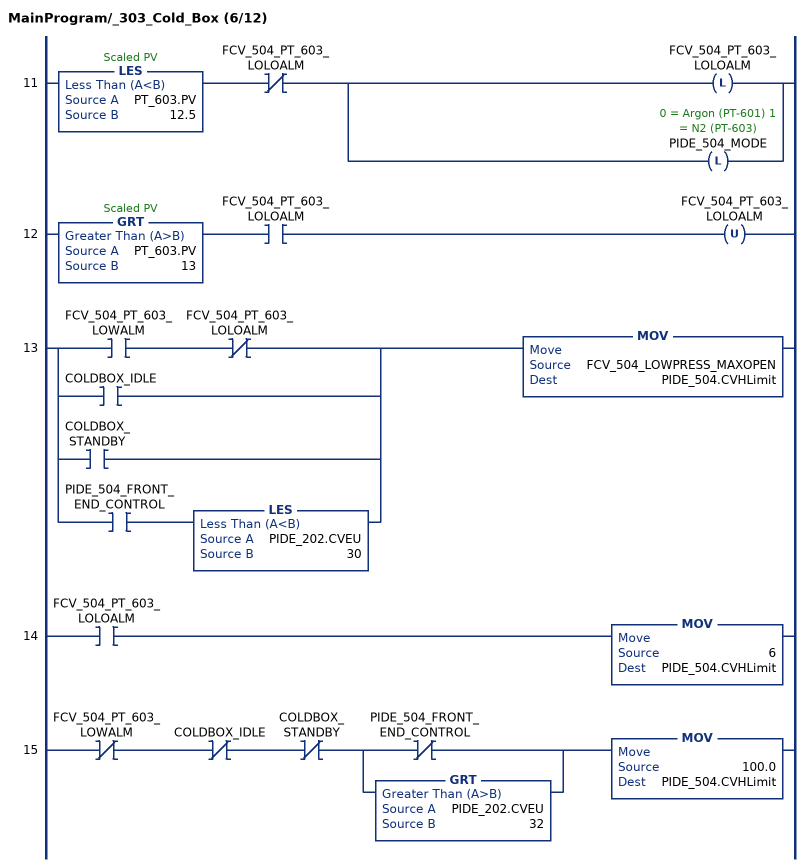
   11: LES(PT_603.PV,12.5)XIO(FCV_504_PT_603_LOLOALM)[OTL(FCV_504_PT_603_LOLOALM) ,OTL(PIDE_504_MODE) ];
   12: GRT(PT_603.PV,13)XIC(FCV_504_PT_603_LOLOALM)OTU(FCV_504_PT_603_LOLOALM);
   13: [XIC(FCV_504_PT_603_LOWALM) XIO(FCV_504_PT_603_LOLOALM) ,XIC(COLDBOX_IDLE) ,XIC(COLDBOX_STANDBY) ,XIC(PIDE_504_FRONT_END_CONTROL) LES(PIDE_202.CVEU,30) ]MOV(FCV_504_LOWPRESS_MAXOPEN,PIDE_504.CVHLimit);
   14: XIC(FCV_504_PT_603_LOLOALM)MOV(6,PIDE_504.CVHLimit);
   15: XIO(FCV_504_PT_603_LOWALM)XIO(COLDBOX_IDLE)XIO(COLDBOX_STANDBY)[XIO(PIDE_504_FRONT_END_CONTROL) ,GRT(PIDE_202.CVEU,32) ]MOV(100.0,PIDE_504.CVHLimit);
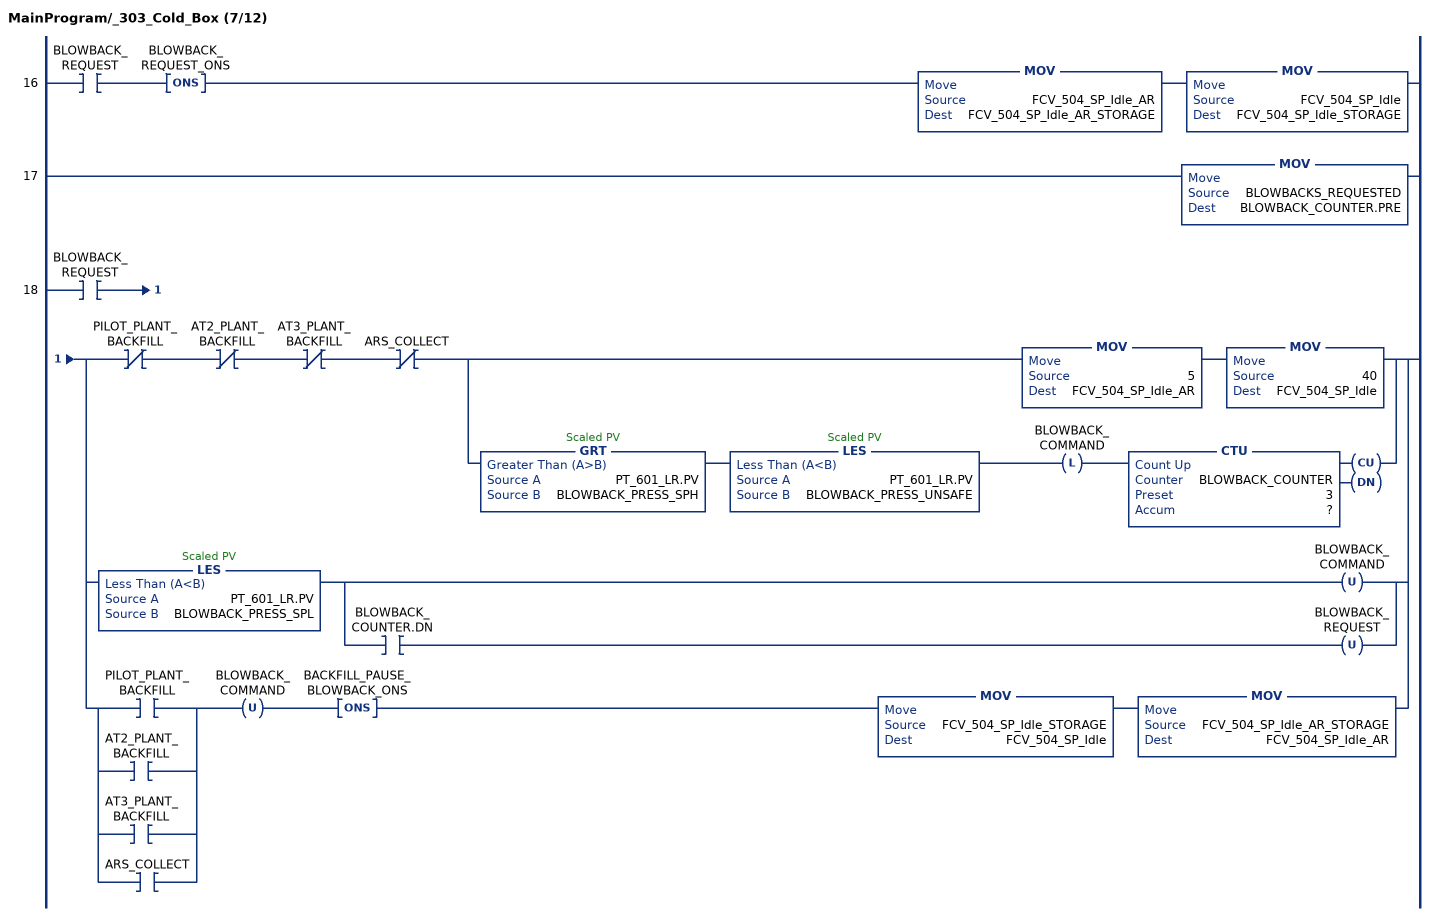
   16: XIC(BLOWBACK_REQUEST)ONS(BLOWBACK_REQUEST_ONS)MOV(FCV_504_SP_Idle_AR,FCV_504_SP_Idle_AR_STORAGE)MOV(FCV_504_SP_Idle,FCV_504_SP_Idle_STORAGE);
   17: MOV(BLOWBACKS_REQUESTED,BLOWBACK_COUNTER.PRE);
   18: XIC(BLOWBACK_REQUEST)[XIO(PILOT_PLANT_BACKFILL) XIO(AT2_PLANT_BACKFILL) XIO(AT3_PLANT_BACKFILL) XIO(ARS_COLLECT) [MOV(5,FCV_504_SP_Idle_AR) MOV(40,FCV_504_SP_Idle) ,GRT(PT_601_LR.PV,BLOWBACK_PRESS_SPH) LES(PT_601_LR.PV,BLOWBACK_PRESS_UNSAFE) OTL(BLOWBACK_COMMAND) CTU(BLOWBACK_COUNTER,?,?) ] ,LES(PT_601_LR.PV,BLOWBACK_PRESS_SPL) [OTU(BLOWBACK_COMMAND) ,XIC(BLOWBACK_COUNTER.DN) OTU(BLOWBACK_REQUEST) ] ,[XIC(PILOT_PLANT_BACKFILL) ,XIC(AT2_PLANT_BACKFILL) ,XIC(AT3_PLANT_BACKFILL) ,XIC(ARS_COLLECT) ] OTU(BLOWBACK_COMMAND) ONS(BACKFILL_PAUSE_BLOWBACK_ONS) MOV(FCV_504_SP_Idle_STORAGE,FCV_504_SP_Idle) MOV(FCV_504_SP_Idle_AR_STORAGE,FCV_504_SP_Idle_AR) ];
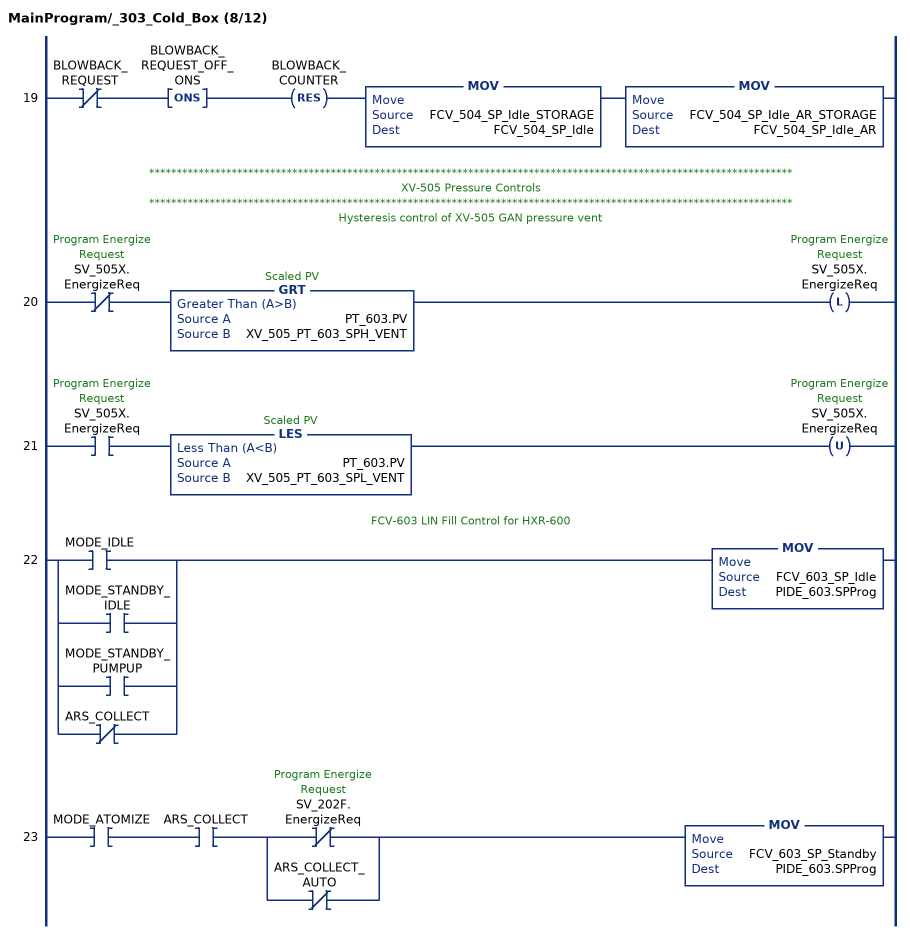
   19: XIO(BLOWBACK_REQUEST)ONS(BLOWBACK_REQUEST_OFF_ONS)RES(BLOWBACK_COUNTER)MOV(FCV_504_SP_Idle_STORAGE,FCV_504_SP_Idle)MOV(FCV_504_SP_Idle_AR_STORAGE,FCV_504_SP_Idle_AR);
   // *********************************************************************************************************************
   // XV-505 Pressure Controls
   // *********************************************************************************************************************
   // Hysteresis control of XV-505 GAN pressure vent
   20: XIO(SV_505X.EnergizeReq)GRT(PT_603.PV,XV_505_PT_603_SPH_VENT)OTL(SV_505X.EnergizeReq);
   21: XIC(SV_505X.EnergizeReq)LES(PT_603.PV,XV_505_PT_603_SPL_VENT)OTU(SV_505X.EnergizeReq);
   // FCV-603 LIN Fill Control for HXR-600
   22: [XIC(MODE_IDLE) ,XIC(MODE_STANDBY_IDLE) ,XIC(MODE_STANDBY_PUMPUP) ,XIO(ARS_COLLECT) ]MOV(FCV_603_SP_Idle,PIDE_603.SPProg);
   23: XIC(MODE_ATOMIZE)XIC(ARS_COLLECT)[XIO(SV_202F.EnergizeReq) ,XIO(ARS_COLLECT_AUTO) ]MOV(FCV_603_SP_Standby,PIDE_603.SPProg);
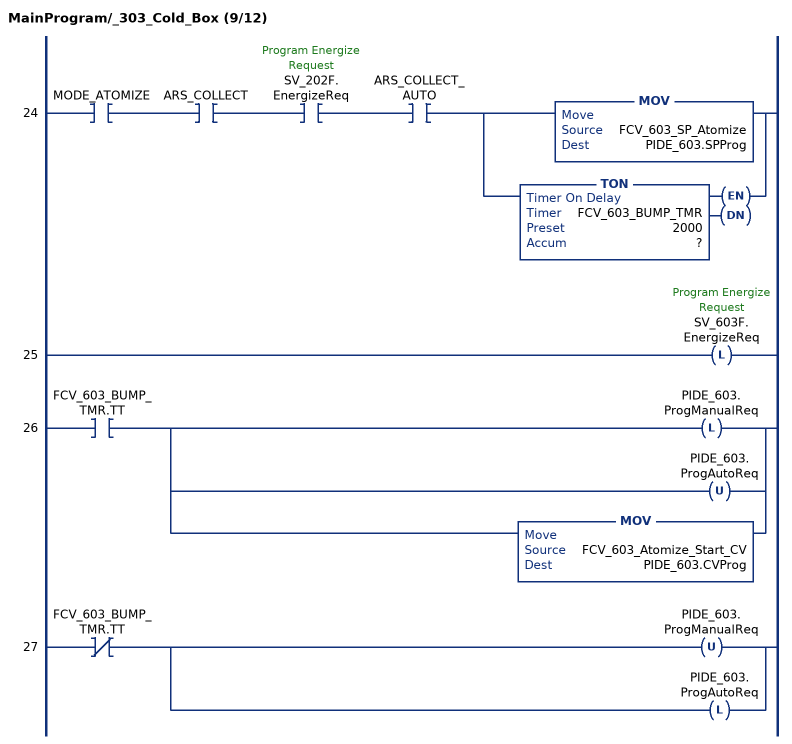
   24: XIC(MODE_ATOMIZE)XIC(ARS_COLLECT)XIC(SV_202F.EnergizeReq)XIC(ARS_COLLECT_AUTO)[MOV(FCV_603_SP_Atomize,PIDE_603.SPProg) ,TON(FCV_603_BUMP_TMR,?,?) ];
   25: OTL(SV_603F.EnergizeReq);
   26: XIC(FCV_603_BUMP_TMR.TT)[OTL(PIDE_603.ProgManualReq) ,OTU(PIDE_603.ProgAutoReq) ,MOV(FCV_603_Atomize_Start_CV,PIDE_603.CVProg) ];
   27: XIO(FCV_603_BUMP_TMR.TT)[OTU(PIDE_603.ProgManualReq) ,OTL(PIDE_603.ProgAutoReq) ];
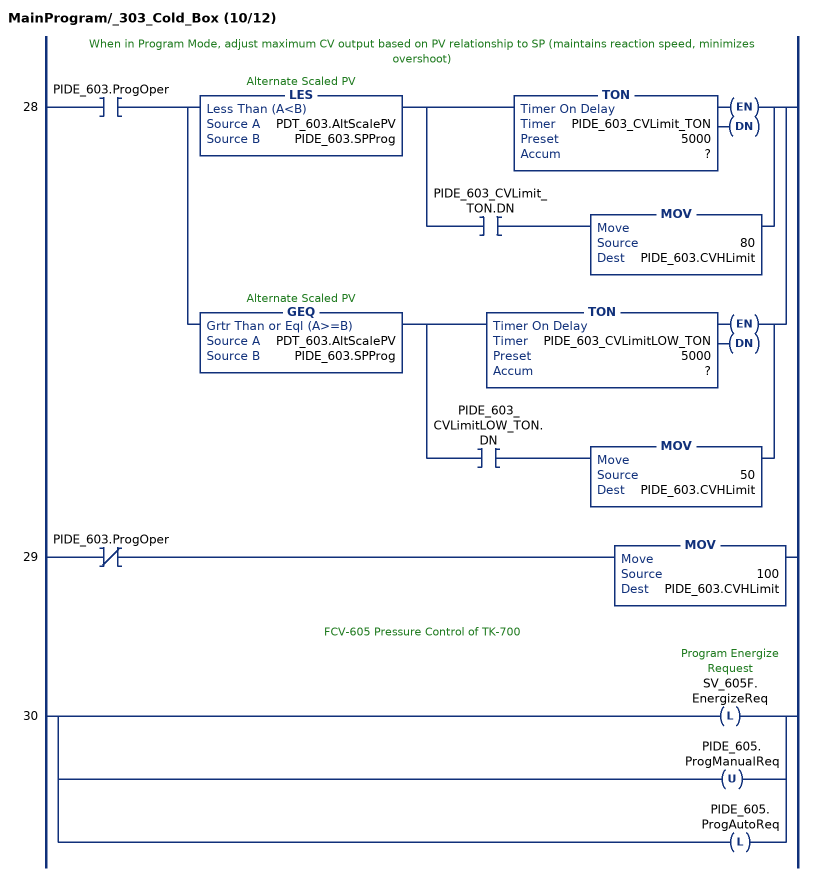
   // When in Program Mode, adjust maximum CV output based on PV relationship to SP (maintains reaction speed, minimizes overshoot)
   28: XIC(PIDE_603.ProgOper)[LES(PDT_603.AltScalePV,PIDE_603.SPProg) [TON(PIDE_603_CVLimit_TON,?,?) ,XIC(PIDE_603_CVLimit_TON.DN) MOV(80,PIDE_603.CVHLimit) ] ,GEQ(PDT_603.AltScalePV,PIDE_603.SPProg) [TON(PIDE_603_CVLimitLOW_TON,?,?) ,XIC(PIDE_603_CVLimitLOW_TON.DN) MOV(50,PIDE_603.CVHLimit) ] ];
   29: XIO(PIDE_603.ProgOper)MOV(100,PIDE_603.CVHLimit);
   // FCV-605 Pressure Control of TK-700
   30: [OTL(SV_605F.EnergizeReq) ,OTU(PIDE_605.ProgManualReq) ,OTL(PIDE_605.ProgAutoReq) ];
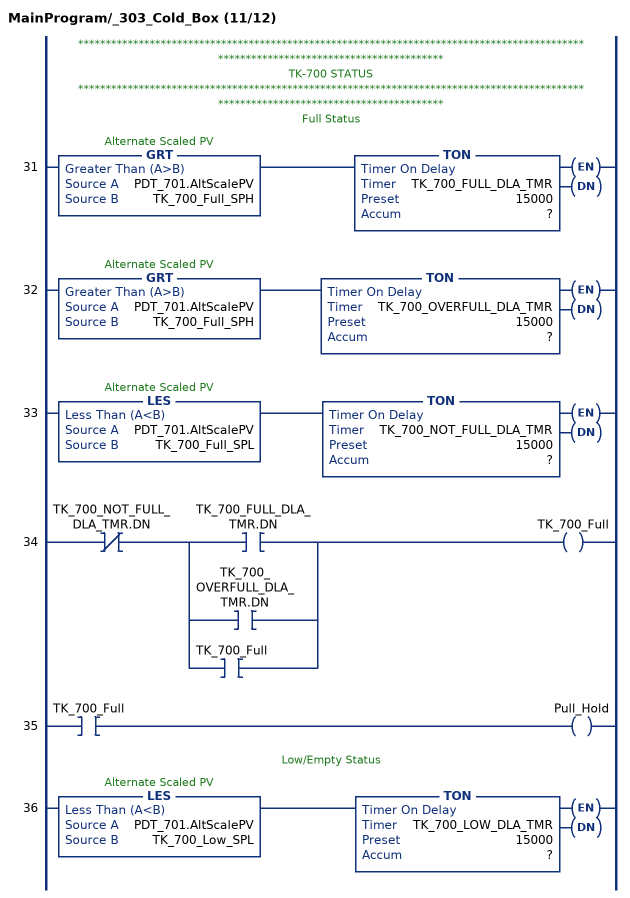
   // *************************************************************************************************************************************
   // TK-700 STATUS
   // *************************************************************************************************************************************
   // Full Status
   31: GRT(PDT_701.AltScalePV,TK_700_Full_SPH)TON(TK_700_FULL_DLA_TMR,?,?);
   32: GRT(PDT_701.AltScalePV,TK_700_Full_SPH)TON(TK_700_OVERFULL_DLA_TMR,?,?);
   33: LES(PDT_701.AltScalePV,TK_700_Full_SPL)TON(TK_700_NOT_FULL_DLA_TMR,?,?);
   34: XIO(TK_700_NOT_FULL_DLA_TMR.DN)[XIC(TK_700_FULL_DLA_TMR.DN) ,XIC(TK_700_OVERFULL_DLA_TMR.DN) ,XIC(TK_700_Full) ]OTE(TK_700_Full);
   35: XIC(TK_700_Full)OTE(Pull_Hold);
   // Low/Empty Status
   36: LES(PDT_701.AltScalePV,TK_700_Low_SPL)TON(TK_700_LOW_DLA_TMR,?,?);
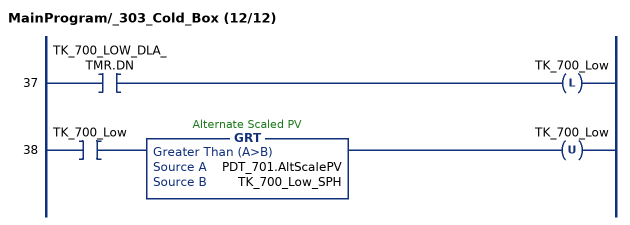
   37: XIC(TK_700_LOW_DLA_TMR.DN)OTL(TK_700_Low);
   38: XIC(TK_700_Low)GRT(PDT_701.AltScalePV,TK_700_Low_SPH)OTU(TK_700_Low);
END_ROUTINE
